# EPICS SNL sequencer program: mcaApp/SISSrc/SIS38XX_SNL.st
program SIS38XX_SNL("P=SIS:3820:, R=mca, NUM_SIGNALS=32,  FIELD=READ")

/*  This sequencer program works with SIS3820.template
 *  It supports multi-element MCA operations
 *
 *  Mark Rivers
 *  April 19, 2011
 *
 * This program must be compiled with the recursive option so that multiple copies
 * can run at once */
option +r;

/* Allow the program to start, even if not all assigned channels are connected.
 * This could be useful if the SNL is running on a different ioc. */
option -c;

%%#include <stdlib.h>
%%#include <errlog.h>
%%#include <string.h>

/* Maximum number of detectors supported */
#define MAX_SIGNALS 32

int i;
int n;
int numSignals;
char temp[100];

char *prefix;
char *record;
char *field;

int   ReadArray[MAX_SIGNALS];
assign  ReadArray to {};
int     ReadArrays; assign ReadArrays to "{P}DoReadAll";
monitor ReadArrays; evflag ReadArraysMon; sync ReadArrays ReadArraysMon;

int     HardwareAcquiring; assign HardwareAcquiring to "{P}HardwareAcquiring";
monitor HardwareAcquiring; evflag HardwareAcquiringMon; sync HardwareAcquiring HardwareAcquiringMon;

int     SNL_Connected;  assign SNL_Connected      to "{P}SNL_Connected";
int     AsynDebug;      assign AsynDebug          to "{P}Asyn.TB1";
monitor AsynDebug;

int Acquiring; assign Acquiring to "{P}Acquiring";

ss mca_control {
  state init {
    when() {
      prefix = macValueGet("P");
      record = macValueGet("R");
      field = macValueGet("FIELD");
      numSignals = atoi(macValueGet("NUM_SIGNALS"));
      if ((numSignals <= 0) || (numSignals > MAX_SIGNALS)) {
        printf ("NUM_SIGNALS is illegal.\n");
        numSignals = 0;
      }
      for (i=0; i<numSignals; i++) {
        n = i+1;
        sprintf(temp, "%s%s%d.%s", prefix, record, n, field);
        pvAssign(ReadArray[i], temp);
       }
    } state waitConnected
  }

  state waitConnected {
    when (numSignals <= 0) {
      printf (">>>>>>>>>>>>>> SIS is dead. <<<<<<<<<<<<<<\n");
    } state dead

    when (pvAssignCount () == pvConnectCount ()) {
      printf ("SIS: All channels connected.\n");
      SNL_Connected = 1;
      pvPut(SNL_Connected);
    } state monitor_changes
  }

  state dead {
    when (delay (3600.0)) {
    } state dead
  }

  state monitor_changes {
    when (pvAssignCount () != pvConnectCount ()) {
      printf ("SIS: Not all channels connected.\n");
    } state waitConnected

    when(efTestAndClear(ReadArraysMon) && (ReadArrays == 1)) {
      if (AsynDebug) printf("SIS.st: Read array data\n");
      for (i=0; i<numSignals; i++) {
        ReadArray[i] = 1;
        pvPut(ReadArray[i]);
      }
      ReadArrays = 0;
      pvPut(ReadArrays);
    } state monitor_changes

    when(efTestAndClear(HardwareAcquiringMon)) {
      if (AsynDebug) printf("SIS.st: HardwareAcquiringMon, HardwareAcquiring=%d\n", HardwareAcquiring);
      /* If the detector is acquiring then force each record to read status */
      if (!HardwareAcquiring) {
        /* If the detector is done then force each record to read data */
        for (i=0; i<numSignals; i++) {
          ReadArray[i] = 1;
          pvPut(ReadArray[i], SYNC);
        }
        /* Clear the Acquiring busy record */
        Acquiring = 0;
        pvPut(Acquiring);
      }
    } state monitor_changes
  }
}
